// TIA Portal V15.1 export
// export: Created 2024-05-17T05:38:26.6840808Z, ExportSetting WithDefaults, DisplayName Totally Integrated Automation Portal, DisplayVersion V15.1 Update 5, DisplayName TIA Portal Openness, DisplayVersion V15.1 Update 5, DisplayName SINAMICS Startdrive Advanced, DisplayVersion V15.1, DisplayName G130, G150, S120, S150, SINAMICS MV, S210, DisplayVersion V15.1, DisplayName G110M, G120, G120C, G120D, G120P, DisplayVersion V15.1, DisplayName STEP 7 Professional, DisplayVersion V15.1 Update 5, DisplayName STEP 7 Safety, DisplayVersion V15.1, DisplayName WinCC Professional, DisplayVersion V15.1 Update 5, DisplayName SIMATIC Visualization Architect, DisplayVersion V15.1
FUNCTION "LInstanceName" : Void   // FC2103, SCL
{ S7_Optimized_Access := 'TRUE' }
VERSION : 0.1
// stored: AutoNumber false, IsIECCheckEnabled false, SetENOAutomatically False, UDAEnableTagReadback false
   VAR_INPUT
      I_GetInstanceName : WString;   // Get Instance Name
   END_VAR
   VAR_OUTPUT
      O_DBName : String;   // DB Name
   END_VAR
   VAR_TEMP
      TmpLEN : Int;
      TmpString : String;
   END_VAR
BEGIN
   #TmpLEN := LEN(#I_GetInstanceName);

   #TmpString := DELETE(IN:=WSTRING_TO_STRING(#I_GetInstanceName), L:=1, P:=#TmpLEN);

   #O_DBName := DELETE(IN := #TmpString, L := 2, P := 1);
END_FUNCTION
